	FUNCTION_BLOCK FB 382
	TITLE =G282M FLAP BOX 9008
	//COPYRIGHT:    (C) 2009  BUHLER AG, CH-9240 UZWIL, SWITZERLAND
	//
	//PRODUCT:      WinCoS_BIW01_09
	//
	//TITLE:        FLAP BOX 9008
	//                Machine group control
	//                Maschinengruppensteuerung
	//
	//--------------------------------------------------------------------------------
	//
	//IDENT:        AUTHOR:             DEPT:                              DATE:
	//
	//P01_FB382.1.0 K.Renz              CSB41                              13.Jan.2010
	//             1st Release
	//
	//--------------------------------------------------------------------------------
	//
	//PURPOSE:
	//
	//MANUAL :
	//
	//RESTRICTIONS:
	//
	//--------------------------------------------------------------------------------
	AUTHOR  : KR
	FAMILY  : USW
	VERSION : 9.9


	VAR
	  Gr       : FB10;	//Standard interface to group
	  InOutValue1    : DINT; //Data for user
	  InOutValue2    : DINT; //Data for user
	  OutWayConflict : BOOL;	//Data for user
	  OutSelectionOk : BOOL;	//Data for user
	  CmdNewValue : BOOL;	//Data for user
	  CmdNewJob   : BOOL;	//Data for user
	  OutCodeOK   : BOOL;	//Data for user
	  InEndOfJob  : BOOL ;	//Data for user
	  staWayOk      : BOOL ;	//Data for user
	  EdgeStartRelease : BOOL ;	//Data for user
	  USW8  : BOOL;	//Data for user
	  USW9 : BOOL;	//Data for user
	  USW10: BOOL;	//Data for user
	  USW11: BOOL;	//Data for user
	  USW12: BOOL;	//Data for user
	  USW13: BOOL;	//Data for user
	  USW14: BOOL;	//Data for user
	  USW15: BOOL;	//Data for user
	     #A_3935_MXZ01_BZS04_05 : FB13;   // VLS
	END_VAR
	VAR_TEMP
	   tmpEnable		: BOOL;
	   tmpFlag  		: BOOL;
	   tmpCmdNext		: BOOL;
	   tmpLocal  		: BOOL;
	   tmpAspOk  		: BOOL;
	   tmpHWStop 		: BOOL;
	   tmpInstanzDBNo       : INT ;
	END_VAR
	BEGIN
	NETWORK
	TITLE =
	NETWORK
	TITLE =Read command from group control
	//Parameter
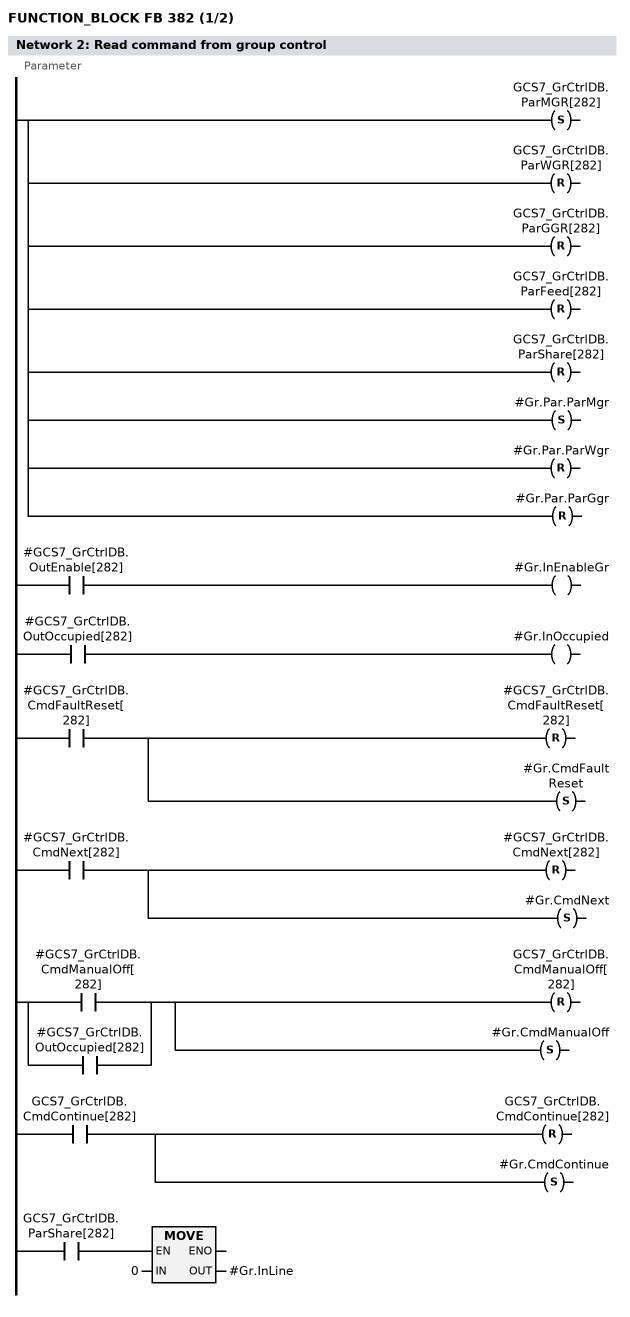
	      SET;
	      S   GCS7_GrCtrlDB.ParMGR[282];
	      R   GCS7_GrCtrlDB.ParWGR[282];
	      R   GCS7_GrCtrlDB.ParGGR[282];
	      R   GCS7_GrCtrlDB.ParFeed[282];
	      R   GCS7_GrCtrlDB.ParShare[282];
	      S   #Gr.Par.ParMgr;
	      R   #Gr.Par.ParWgr;
	      R   #Gr.Par.ParGgr;
	//Command
	      U   #GCS7_GrCtrlDB.OutEnable[282];
	      =   #Gr.InEnableGr;
	      U   #GCS7_GrCtrlDB.OutOccupied[282];
	      =   #Gr.InOccupied;
	      U   #GCS7_GrCtrlDB.CmdFaultReset[282];
	      R   #GCS7_GrCtrlDB.CmdFaultReset[282];
	      S   #Gr.CmdFaultReset;
	      U  #GCS7_GrCtrlDB.CmdNext[282];
	      R   #GCS7_GrCtrlDB.CmdNext[282];
	      S   #Gr.CmdNext;
	      U   #GCS7_GrCtrlDB.CmdManualOff[282];
	      O   #GCS7_GrCtrlDB.OutOccupied[282];
	      R   GCS7_GrCtrlDB.CmdManualOff[282];
	      S   #Gr.CmdManualOff;
	      U  GCS7_GrCtrlDB.CmdContinue[282];
	      R   GCS7_GrCtrlDB.CmdContinue[282];
	      S   #Gr.CmdContinue;
	//Init Line Number
	      U   GCS7_GrCtrlDB.ParShare[282];
	      SPBN WE00;
	      L     0;
	      T     #Gr.InLine;
	WE00: NOP   0;
	NETWORK
	TITLE =Call Methode Control
	// 1. Handle Interface PCControl
	// 2. Prepare mode --> ModePassive,ModeActive,ModeIdling
	// 3. Reset global flags of the group
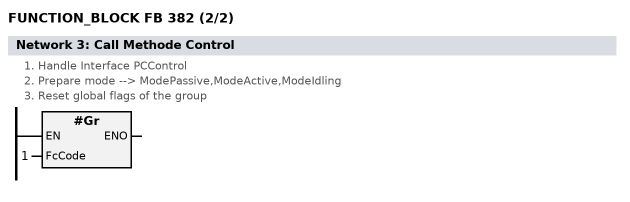
	      CALL #Gr (
	           FcCode                   := 1);
	NETWORK
	TITLE =Restart Idling Time
		L  #Gr.Par.ParIdling;
		L  2;
		>=I;
		SPB IdTm;
		T  #Gr.Par.ParIdling;
	IdTm:   NOP 0;
	      CLR;
	      S    #Gr.CmdRestartIdling;
	NETWORK
	TITLE =Prepare global flags
	NETWORK
	TITLE =Set Pattern (Target position)
	NETWORK
	TITLE =Interlocking WayOk
	//
	NETWORK
	TITLE =Interlocking Autostart
		CLR;
		R   #Gr.OutAutostart;
	NETWORK
	TITLE =Interlocking Enable
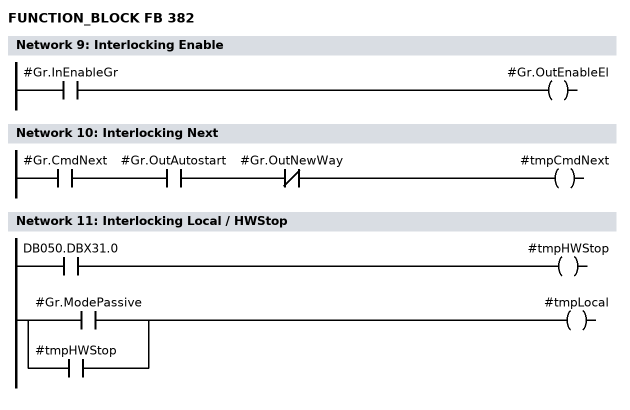
	      U     #Gr.InEnableGr;
	      =     #Gr.OutEnableEl;

	NETWORK
	TITLE =Interlocking Next
	      U     #Gr.CmdNext;
	      U     #Gr.OutAutostart;
	      UN    #Gr.OutNewWay;
	      =    #tmpCmdNext;

	NETWORK
	TITLE =Interlocking Local / HWStop
	      U    DB050.DBX31.0;
	      =    #tmpHWStop;

	      U    #Gr.ModePassive;
	      O    #tmpHWStop;
	      =    #tmpLocal;

	NETWORK
	TITLE ==A-3935-MXZ01/BZS04/05 : FLAP BOX 9008
	NOP 0;
	//-InLocal---
	      U     #tmpLocal;
	      =     #A_3935_MXZ01_BZS04_05.InLocal;
	//
	//-Interlocking---
	         =     #A_3935_MXZ01_BZS04_05.InEnableHN;
	         NOT;
	         =     #A_3935_MXZ01_BZS04_05.InEnableLN;
	//
	         SET;
	         S     #A_3935_MXZ01_BZS04_05.CmdNext;
	//
	      U     #Gr.OutSeqStop;
	      =     #A_3935_MXZ01_BZS04_05.InSeqStop;
	//
	//-Read inputs---
	      U     E 1138.0;
	      =     #A_3935_MXZ01_BZS04_05.InpLN;
	      U     E 1138.1;
	      =     #A_3935_MXZ01_BZS04_05.InpHN;
	      X     A 1135.2;
	      X     E 1135.2;
	      O;
	      X     A 1135.3;
	      X     E 1135.3;
	      =     #A_3935_MXZ01_BZS04_05.InpFaultDev;
	      U   DB050.DBX32.5;
	      =     #A_3935_MXZ01_BZS04_05.InHWStop;
	       U     PLC_DPInfo.Master[1].SlavesError[114];
	       =       #A_3935_MXZ01_BZS04_05.InDPFault;
	//
	//-Set Parameters---
	//
	//-Call object control---
	      CALL  #A_3935_MXZ01_BZS04_05;
	//
	//-Write outputs---
	      U     #A_3935_MXZ01_BZS04_05.OutpLN;
	      =     A 1135.2;
	      U     #A_3935_MXZ01_BZS04_05.OutpHN;
	      =     A 1135.3;
	NETWORK
	TITLE =Test Fault
	      U     #A_3935_MXZ01_BZS04_05.StFault;
	      =     #Gr.VarFault;
	NETWORK
	TITLE =Test Warning
	      CLR;
	      =     #Gr.OutWarning;
	NETWORK
	TITLE =Test Stopped
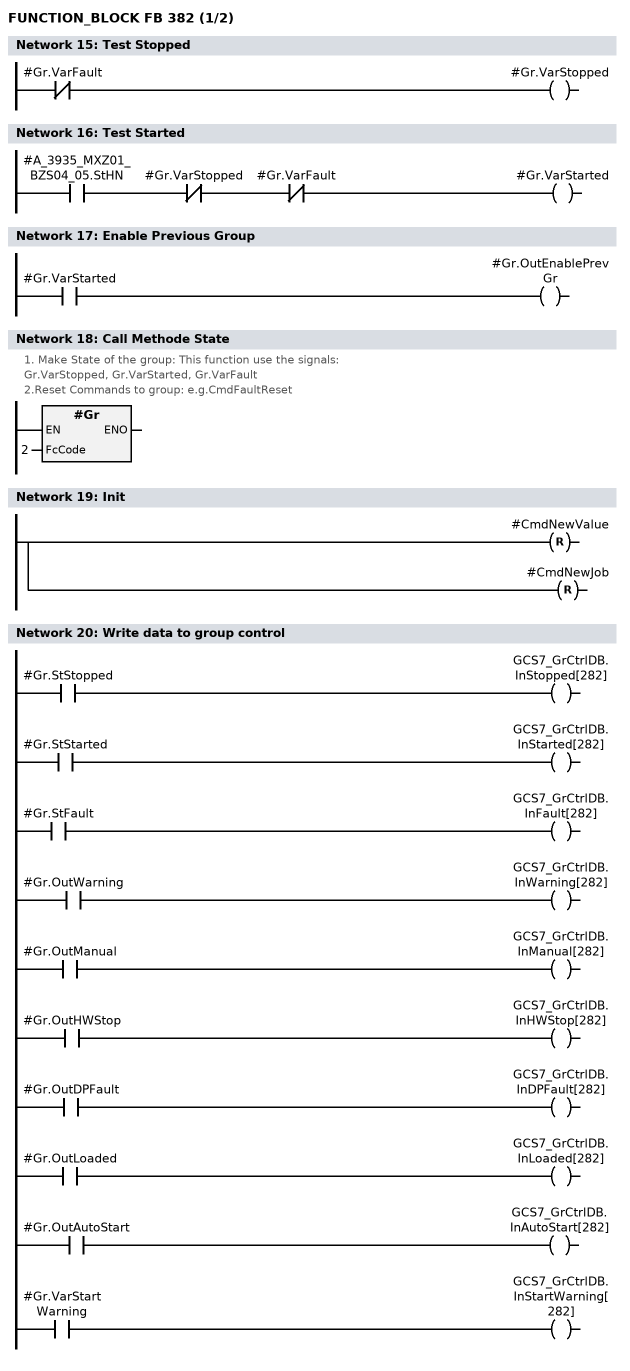
	      UN   #Gr.VarFault;
	      =     #Gr.VarStopped;
	NETWORK
	TITLE =Test Started
	      U     #A_3935_MXZ01_BZS04_05.StHN;
	      UN  #Gr.VarStopped;
	      UN  #Gr.VarFault;
	      =     #Gr.VarStarted;
	NETWORK
	TITLE =Enable Previous Group
	      U    #Gr.VarStarted;
	      =     #Gr.OutEnablePrevGr;
	NETWORK
	TITLE =Call Methode State
	//1. Make State of the group: This function use the signals:
	//        Gr.VarStopped, Gr.VarStarted, Gr.VarFault
	//2.Reset Commands to group: e.g.CmdFaultReset
	      CALL #Gr (
	           FcCode                   := 2);
	NETWORK
	TITLE =Init
	      SET;
	      R    #CmdNewValue;
	      R    #CmdNewJob;
	NETWORK
	TITLE =Write data to group control
	      U   #Gr.StStopped;
	      =   GCS7_GrCtrlDB.InStopped[282];
	      U   #Gr.StStarted;
	      =   GCS7_GrCtrlDB.InStarted[282];
	      U   #Gr.StFault;
	      =   GCS7_GrCtrlDB.InFault[282];
	      U   #Gr.OutWarning;
	      =   GCS7_GrCtrlDB.InWarning[282];
	      U   #Gr.OutManual;
	      =   GCS7_GrCtrlDB.InManual[282];
	      U   #Gr.OutHWStop;
	      =   GCS7_GrCtrlDB.InHWStop[282];
	      U   #Gr.OutDPFault;
	      =   GCS7_GrCtrlDB.InDPFault[282];
	      U   #Gr.OutLoaded;
	      =   GCS7_GrCtrlDB.InLoaded[282];
	      U   #Gr.OutAutoStart;
	      =   GCS7_GrCtrlDB.InAutoStart[282];
	      U   #Gr.VarStartWarning;
	      =   GCS7_GrCtrlDB.InStartWarning[282];
	NETWORK
	TITLE =End of block
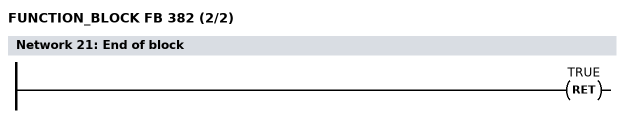

	BE

	END_FUNCTION_BLOCK
